{attribute 'pack_mode' := '1'}
TYPE ST_CloseShutter EXTENDS ST_MsgToPLC:
STRUCT

END_STRUCT
END_TYPE

(* stored: Version 1.1.0.1, ProductVersion 3.1.4022.18
   DUT ST_CloseShutter: Id {810fd15a-843a-4824-afc1-ec18e84cc650} *)
